TYPE ST_BleutoothControl :
STRUCT
	EnableBleutoothDiagnosis	: BOOL;
	ActivatePairingMode			: BOOL;
END_STRUCT
END_TYPE

(* stored: Version 1.1.0.1
   DUT ST_BleutoothControl: Id {f1b73aa4-1f95-4fe5-8fe0-b057c116e6c5} *)
